FUNCTION_BLOCK FB_AxisBase IMPLEMENTS ITF_Base
VAR_INPUT
END_VAR
VAR_OUTPUT
END_VAR
VAR
	_axis : AXIS_REF;
	_power : MC_Power;
	_reset : MC_Reset;
	_status : ST_AxisStatus;
	_override : LREAL;
	_enableNegativeDirection : BOOL;
	_enabled : BOOL;
END_VAR

_power(Axis := _axis);
_reset(Axis := _axis);
_status := GetStatus();

METHOD PUBLIC Disable : BOOL
VAR_INPUT
END_VAR
IF NOT _power.Status THEN
	Disable := TRUE;
	_enabled := FALSE;
ELSE
	_power.Enable := FALSE;
END_IF
END_METHOD

METHOD PUBLIC Enable : BOOL
VAR_INPUT
END_VAR
IF (_power.Status) THEN
	Enable := TRUE;
	_enabled := TRUE;
ELSE
	_power.Enable := TRUE;
	_power.Enable_Negative := _enableNegativeDirection;
	_power.Enable_Positive := TRUE;
	_power.Override := _override;
END_IF
END_METHOD

PROPERTY PUBLIC Enabled : bool
GET
Enabled := _enabled;
END_GET
END_PROPERTY

{warning 'add property implementation'}
PROPERTY EnableNegativeDirection : BOOL
GET
EnableNegativeDirection := _enableNegativeDirection;
END_GET
SET
_enableNegativeDirection := EnableNegativeDirection;
END_SET
END_PROPERTY

METHOD PROTECTED GetStatus : st_AxisStatus
VAR_INPUT
END_VAR
_axis.ReadStatus();
GetStatus := _axis.Status;
END_METHOD

{warning 'add property implementation'}
PROPERTY Override : LREAL
GET
Override := _override;
END_GET
SET
_override := Override;
END_SET
END_PROPERTY

METHOD PUBLIC Reset : BOOL
VAR_INPUT
END_VAR
_reset.Execute := TRUE;
IF _reset.Done AND NOT _reset.Error THEN
	Reset := TRUE;
END_IF
END_METHOD

END_FUNCTION_BLOCK

(* stored: Version 1.1.0.1, ProductVersion 3.1.4024.3
   POU FB_AxisBase: Id {dbf7b8f1-ae81-4287-be87-eea1c81c44ed}, SpecialFunc None
   Folder Functions: Id {fa1131cc-8ce1-4d4a-ae8f-5bfb26f51f70}
   Folder Properties: Id {3f341a9f-4117-4254-8d8b-3dba578ac155}
   Method Disable: Id {1e1f04b1-019f-447e-9dae-9f9045650318}
   Method Enable: Id {db2ed9b3-ee26-4fe1-966d-2deb43f58bd6}
   Property Enabled: Id {5632354a-4462-4802-be31-68adbf70f687}
   Get Get: Id {438cd9c9-cfc0-463c-a089-72c0119c0d70}
   Property EnableNegativeDirection: Id {fec7bd58-0f65-4325-8cb9-d508f03f0c9f}
   Get Get: Id {cf9e60e9-91e1-4213-a3db-cb0cd7337eb8}
   Set Set: Id {410ae65e-bdaf-49c2-b8dd-de0099ba81ce}
   Method GetStatus: Id {247164c8-fa59-429a-8f8b-9799cf350735}
   Property Override: Id {ed9bd1fd-b6a2-4b9c-995d-0becc00f218f}
   Get Get: Id {0accf564-84f3-4f9d-b305-14de34ae3804}
   Set Set: Id {e8ddcebe-6280-4196-af0c-edff922a562c}
   Method Reset: Id {2ad1e6d6-18b8-4736-81d3-000694ff865a} *)
